INTERFACE ITask

METHOD Abort : BOOL
VAR_INPUT
END_VAR
END_METHOD

PROPERTY Busy : bool
GET
END_GET
END_PROPERTY

PROPERTY Done : bool
GET
END_GET
END_PROPERTY

PROPERTY Error : bool
GET
END_GET
END_PROPERTY

METHOD Execute : BOOL
VAR_INPUT
END_VAR
END_METHOD

END_INTERFACE

(* stored: Version 1.1.0.1, ProductVersion 3.1.4024.11
   Itf ITask: Id {65c388f3-e60b-4c18-859b-50e2fcc598a3}
   Method Abort: Id {5fbeff62-a4be-4548-9a99-67f58198dc76}
   Property Busy: Id {5998b8c2-c47f-436c-8aef-3dae2966b3dd}
   Get Get: Id {12b78287-799e-43ac-aa6e-b101486bd11a}
   Property Done: Id {cae6d50e-a879-4668-8186-fe39c41c78ad}
   Get Get: Id {3a84c623-4709-4ee2-9c11-f1e9b211716e}
   Property Error: Id {6c03825f-ff37-4bbd-b166-7f80e077ca72}
   Get Get: Id {683df8b9-fb69-428d-b622-2208d2e75585}
   Method Execute: Id {783a8a72-0411-4f1e-8388-2cce2298d54a} *)
